PROGRAM MAIN
VAR
	_technology : Technology;
END_VAR

_technology.Run();

END_PROGRAM

(* stored: Version 1.1.0.1, ProductVersion 3.1.4024.9
   POU MAIN: Id {59823e5a-7765-4e6b-9b38-dce68759b26f}, SpecialFunc None *)
